// TIA Portal V16 export
// export: Created 2022-07-21T09:35:34.8398249Z, ExportSetting WithDefaults, DisplayName Totally Integrated Automation Portal, DisplayVersion V16 Update 4, DisplayName TIA Portal Version Control Interface, DisplayVersion V16 Update 2, DisplayName TIA Portal Openness, DisplayVersion V16 Update 4, DisplayName SINAMICS Startdrive Advanced, DisplayVersion V16 Update 5, DisplayName SINAMICS Startdrive G130, G150, S120, S150, SINAMICS MV, S210, DisplayVersion V16 Update 5, DisplayName SINAMICS Startdrive G110M, G120, G120C, G120D, G120P, G115D, DisplayVersion V16 Update 5, DisplayName STEP 7 Professional, DisplayVersion V16 Update 4, DisplayName STEP 7 Safety, DisplayVersion V16, DisplayName WinCC Advanced, DisplayVersion V16 Update 4
FUNCTION_BLOCK "fbGroup"   // FB700, LAD
TITLE = Group / Grupa
{ S7_Optimized_Access := 'TRUE' }
VERSION : 0.1
// stored: AutoNumber false, IsIECCheckEnabled false, IsRetainMemResEnabled false, MemoryReserve 100, SetENOAutomatically false, UDAEnableTagReadback false
   VAR_INPUT
      startDelay : Time := T#1s;   // Czas opóźnienia dla startu grupy / Start delay
      cancelEndOfSeq : Bool;   // Sygnał anulowania zatrzymania na końcu sekwencji / Cancel stop end of sequence
   END_VAR
   VAR_OUTPUT
      startup : Bool;   // Ostrzeżenie przed uruchomieniem pracy w trybie auto / Warning startup in automatic mode
   END_VAR
   VAR_IN_OUT
      group : "typeGroup";   // Grupa / Group
      extGroup : "typeGroup";   // Żądanie zewnętrzne / External request
   END_VAR
   VAR
      instTmrDlyStart { S7_SetPoint := 'True'} : TON_TIME;   // Opóźnienie dla startu grupy / Start delay
      instReset { S7_SetPoint := 'True'} : "fbReset";
      statPManual { S7_SetPoint := 'True'} : Bool;
      statPStep : Bool;
      statPAuto : Bool;
      statNSafe : Bool;
      instTmrHomeCmd { S7_SetPoint := 'True'} : TON_TIME;
   END_VAR
   VAR_TEMP   // added for the SCL form of the ladder/FBD networks
      _w1 : Bool;
      _w2 : Bool;
   END_VAR
BEGIN

REGION Network 1: Komenda "Reset"
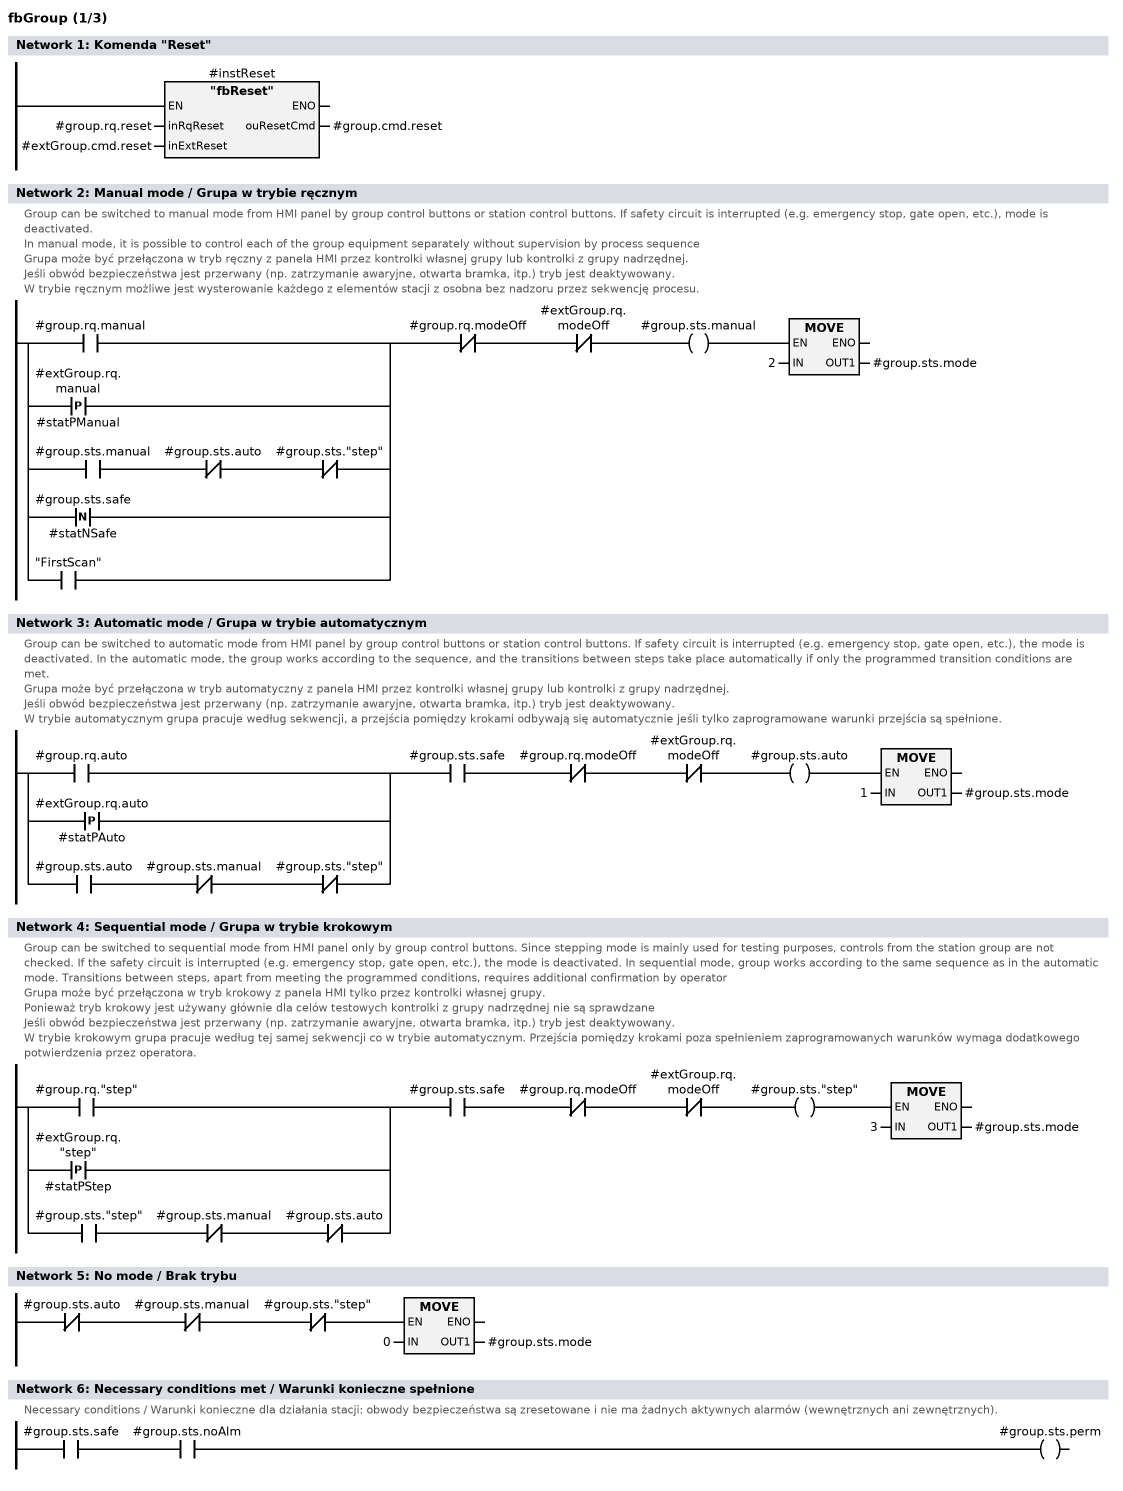
   RUNG wire#powerrail
      #instReset(inRqReset := #group.rq.reset, inExtReset := #extGroup.cmd.reset, ouResetCmd => #group.cmd.reset)
   END_RUNG
   // the same network as SCL:
   #instReset(inRqReset := #group.rq.reset, inExtReset := #extGroup.cmd.reset, ouResetCmd => #group.cmd.reset);   // "fbReset"
END_REGION

REGION Network 2: Manual mode / Grupa w trybie ręcznym
   // Group can be switched to manual mode from HMI panel by group control buttons or station control buttons. If safety circuit is interrupted (e.g. emergency stop, gate open, etc.), mode is deactivated.
   //  In manual mode, it is possible to control each of the group equipment separately without supervision by process sequence
   // Grupa może być przełączona w tryb ręczny z panela HMI przez kontrolki własnej grupy lub kontrolki z grupy nadrzędnej.
   // Jeśli obwód bezpieczeństwa jest przerwany (np. zatrzymanie awaryjne, otwarta bramka, itp.) tryb jest deaktywowany.
   // W trybie ręcznym możliwe jest wysterowanie każdego z elementów stacji z osobna bez nadzoru przez sekwencję procesu.
   RUNG wire#powerrail
      Contact( #group.rq.manual )
      wire#w1
      I_Contact( #group.rq.modeOff )
      I_Contact( #extGroup.rq.modeOff )
      Coil( #group.sts.manual )
      Move(in := 2, out1 => #group.sts.mode)
   END_RUNG
   RUNG wire#powerrail
      P_Contact(operand := #extGroup.rq.manual, bit := #statPManual)
   END_RUNG wire#w1
   RUNG wire#powerrail
      Contact( #group.sts.manual )
      I_Contact( #group.sts.auto )
      I_Contact( #group.sts."step" )
   END_RUNG wire#w1
   RUNG wire#powerrail
      N_Contact(operand := #group.sts.safe, bit := #statNSafe)
   END_RUNG wire#w1
   RUNG wire#powerrail
      Contact( "FirstScan" )
   END_RUNG wire#w1
   // the same network as SCL:
   #_w1 := #extGroup.rq.manual AND NOT #statPManual;   // rising edge of #extGroup.rq.manual
   #statPManual := #extGroup.rq.manual;
   #_w2 := NOT #group.sts.safe AND #statNSafe;   // falling edge of #group.sts.safe
   #statNSafe := #group.sts.safe;
   #group.sts.manual := (#group.rq.manual OR #_w1 OR (#group.sts.manual AND NOT #group.sts.auto AND NOT #group.sts."step") OR #_w2 OR "FirstScan") AND NOT #group.rq.modeOff AND NOT #extGroup.rq.modeOff;
   IF #group.sts.manual THEN #group.sts.mode := 2; END_IF;
END_REGION

REGION Network 3: Automatic mode / Grupa w trybie automatycznym
   // Group can be switched to automatic mode from HMI panel by group control buttons or station control buttons. If safety circuit is interrupted (e.g. emergency stop, gate open, etc.), the mode is deactivated. In the automatic mode, the group works according to the sequence, and the transitions between steps take place automatically if only the programmed transition conditions are met.
   // Grupa może być przełączona w tryb automatyczny z panela HMI przez kontrolki własnej grupy lub kontrolki z grupy nadrzędnej.
   // Jeśli obwód bezpieczeństwa jest przerwany (np. zatrzymanie awaryjne, otwarta bramka, itp.) tryb jest deaktywowany.
   // W trybie automatycznym grupa pracuje według sekwencji, a przejścia pomiędzy krokami odbywają się automatycznie jeśli tylko zaprogramowane warunki przejścia są spełnione.
   RUNG wire#powerrail
      Contact( #group.rq.auto )
      wire#w1
      Contact( #group.sts.safe )
      I_Contact( #group.rq.modeOff )
      I_Contact( #extGroup.rq.modeOff )
      Coil( #group.sts.auto )
      Move(in := 1, out1 => #group.sts.mode)
   END_RUNG
   RUNG wire#powerrail
      P_Contact(operand := #extGroup.rq.auto, bit := #statPAuto)
   END_RUNG wire#w1
   RUNG wire#powerrail
      Contact( #group.sts.auto )
      I_Contact( #group.sts.manual )
      I_Contact( #group.sts."step" )
   END_RUNG wire#w1
   // the same network as SCL:
   #_w1 := #extGroup.rq.auto AND NOT #statPAuto;   // rising edge of #extGroup.rq.auto
   #statPAuto := #extGroup.rq.auto;
   #group.sts.auto := (#group.rq.auto OR #_w1 OR (#group.sts.auto AND NOT #group.sts.manual AND NOT #group.sts."step")) AND #group.sts.safe AND NOT #group.rq.modeOff AND NOT #extGroup.rq.modeOff;
   IF #group.sts.auto THEN #group.sts.mode := 1; END_IF;
END_REGION

REGION Network 4: Sequential mode / Grupa w trybie krokowym
   // Group can be switched to sequential mode from HMI panel only by group control buttons. Since stepping mode is mainly used for testing purposes, controls from the station group are not checked. If the safety circuit is interrupted (e.g. emergency stop, gate open, etc.), the mode is deactivated. In sequential mode, group works according to the same sequence as in the automatic mode. Transitions between steps, apart from meeting the programmed conditions, requires additional confirmation by operator
   // Grupa może być przełączona w tryb krokowy z panela HMI tylko przez kontrolki własnej grupy.
   // Ponieważ tryb krokowy jest używany głównie dla celów testowych kontrolki z grupy nadrzędnej nie są sprawdzane
   // Jeśli obwód bezpieczeństwa jest przerwany (np. zatrzymanie awaryjne, otwarta bramka, itp.) tryb jest deaktywowany.
   // W trybie krokowym grupa pracuje według tej samej sekwencji co w trybie automatycznym. Przejścia pomiędzy krokami poza spełnieniem zaprogramowanych warunków wymaga dodatkowego potwierdzenia przez operatora.
   RUNG wire#powerrail
      Contact( #group.rq."step" )
      wire#w1
      Contact( #group.sts.safe )
      I_Contact( #group.rq.modeOff )
      I_Contact( #extGroup.rq.modeOff )
      Coil( #group.sts."step" )
      Move(in := 3, out1 => #group.sts.mode)
   END_RUNG
   RUNG wire#powerrail
      P_Contact(operand := #extGroup.rq."step", bit := #statPStep)
   END_RUNG wire#w1
   RUNG wire#powerrail
      Contact( #group.sts."step" )
      I_Contact( #group.sts.manual )
      I_Contact( #group.sts.auto )
   END_RUNG wire#w1
   // the same network as SCL:
   #_w1 := #extGroup.rq."step" AND NOT #statPStep;   // rising edge of #extGroup.rq."step"
   #statPStep := #extGroup.rq."step";
   #group.sts."step" := (#group.rq."step" OR #_w1 OR (#group.sts."step" AND NOT #group.sts.manual AND NOT #group.sts.auto)) AND #group.sts.safe AND NOT #group.rq.modeOff AND NOT #extGroup.rq.modeOff;
   IF #group.sts."step" THEN #group.sts.mode := 3; END_IF;
END_REGION

REGION Network 5: No mode / Brak trybu
   RUNG wire#powerrail
      I_Contact( #group.sts.auto )
      I_Contact( #group.sts.manual )
      I_Contact( #group.sts."step" )
      Move(in := 0, out1 => #group.sts.mode)
   END_RUNG
   // the same network as SCL:
   IF NOT #group.sts.auto AND NOT #group.sts.manual AND NOT #group.sts."step" THEN
       #group.sts.mode := 0;
   END_IF;
END_REGION

REGION Network 6: Necessary conditions met / Warunki konieczne spełnione
   // Necessary conditions / Warunki konieczne dla działania stacji: obwody bezpieczeństwa są zresetowane i nie ma żadnych aktywnych alarmów (wewnętrznych ani zewnętrznych).
   RUNG wire#powerrail
      Contact( #group.sts.safe )
      Contact( #group.sts.noAlm )
      Coil( #group.sts.perm )
   END_RUNG
   // the same network as SCL:
   #group.sts.perm := #group.sts.safe AND #group.sts.noAlm;
END_REGION

REGION Network 7: Ready to start / Grupa gotowa do startu
   // Group is ready to start if automatic/sequential mode is selected, necessary conditions are met, all equipment is in home position, sequence is in initial step / Grupa jest gotowa do rozpoczęcia pracy według sekwencji jeśli wybrano tryb automatyczny lub krokowy, warunki konieczne są spełnione, wszystkie elementy stacji są w pozycji bazowej i sekwencja pracy znajduje się w kroku początkowym.
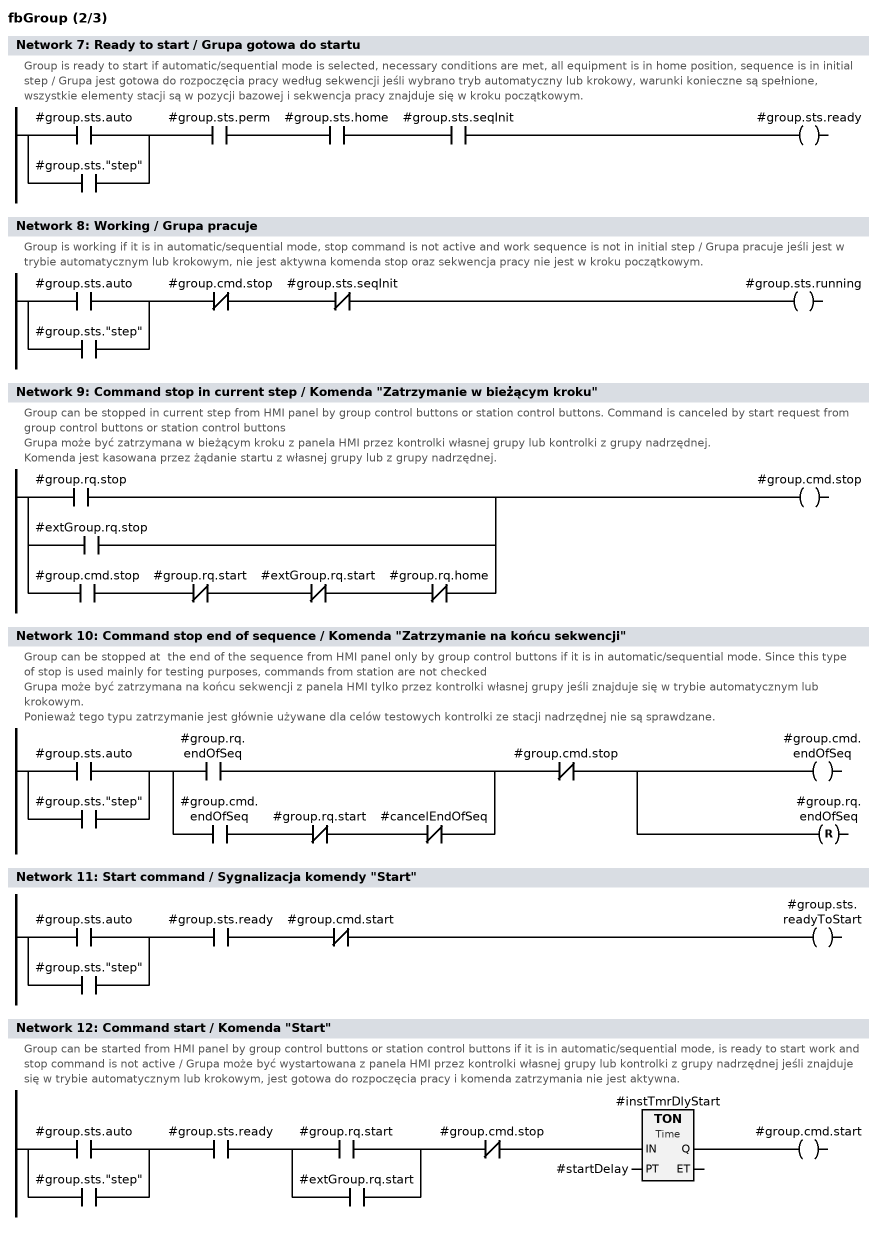
   RUNG wire#powerrail
      Contact( #group.sts.auto )
      wire#w1
      Contact( #group.sts.perm )
      Contact( #group.sts.home )
      Contact( #group.sts.seqInit )
      Coil( #group.sts.ready )
   END_RUNG
   RUNG wire#powerrail
      Contact( #group.sts."step" )
   END_RUNG wire#w1
   // the same network as SCL:
   #group.sts.ready := (#group.sts.auto OR #group.sts."step") AND #group.sts.perm AND #group.sts.home AND #group.sts.seqInit;
END_REGION

REGION Network 8: Working / Grupa pracuje
   // Group is working if it is in automatic/sequential mode, stop command is not active and work sequence is not in initial step / Grupa pracuje jeśli jest w trybie automatycznym lub krokowym, nie jest aktywna komenda stop oraz sekwencja pracy nie jest w kroku początkowym.
   RUNG wire#powerrail
      Contact( #group.sts.auto )
      wire#w1
      I_Contact( #group.cmd.stop )
      I_Contact( #group.sts.seqInit )
      Coil( #group.sts.running )
   END_RUNG
   RUNG wire#powerrail
      Contact( #group.sts."step" )
   END_RUNG wire#w1
   // the same network as SCL:
   #group.sts.running := (#group.sts.auto OR #group.sts."step") AND NOT #group.cmd.stop AND NOT #group.sts.seqInit;
END_REGION

REGION Network 9: Command stop in current step / Komenda "Zatrzymanie w bieżącym kroku"
   // Group can be stopped in current step from HMI panel by group control buttons or station control buttons. Command is canceled by start request from group control buttons or station control buttons
   // Grupa może być zatrzymana w bieżącym kroku z panela HMI przez kontrolki własnej grupy lub kontrolki z grupy nadrzędnej.
   // Komenda jest kasowana przez żądanie startu z własnej grupy lub z grupy nadrzędnej.
   RUNG wire#powerrail
      Contact( #group.rq.stop )
      wire#w1
      Coil( #group.cmd.stop )
   END_RUNG
   RUNG wire#powerrail
      Contact( #extGroup.rq.stop )
   END_RUNG wire#w1
   RUNG wire#powerrail
      Contact( #group.cmd.stop )
      I_Contact( #group.rq.start )
      I_Contact( #extGroup.rq.start )
      I_Contact( #group.rq.home )
   END_RUNG wire#w1
   // the same network as SCL:
   #group.cmd.stop := #group.rq.stop OR #extGroup.rq.stop OR (#group.cmd.stop AND NOT #group.rq.start AND NOT #extGroup.rq.start AND NOT #group.rq.home);
END_REGION

REGION Network 10: Command stop end of sequence / Komenda "Zatrzymanie na końcu sekwencji"
   // Group can be stopped at  the end of the sequence from HMI panel only by group control buttons if it is in automatic/sequential mode. Since this type of stop is used mainly for testing purposes, commands from station are not checked
   // Grupa może być zatrzymana na końcu sekwencji z panela HMI tylko przez kontrolki własnej grupy jeśli znajduje się w trybie automatycznym lub krokowym.
   // Ponieważ tego typu zatrzymanie jest głównie używane dla celów testowych kontrolki ze stacji nadrzędnej nie są sprawdzane.
   RUNG wire#powerrail
      Contact( #group.sts.auto )
      wire#w1
      Contact( #group.rq.endOfSeq )
      wire#w2
      I_Contact( #group.cmd.stop )
      wire#w3
      Coil( #group.cmd.endOfSeq )
   END_RUNG
   RUNG wire#powerrail
      Contact( #group.sts."step" )
   END_RUNG wire#w1
   RUNG wire#w1
      Contact( #group.cmd.endOfSeq )
      I_Contact( #group.rq.start )
      I_Contact( #cancelEndOfSeq )
   END_RUNG wire#w2
   RUNG wire#w3
      R_Coil( #group.rq.endOfSeq )
   END_RUNG
   // the same network as SCL:
   #group.cmd.endOfSeq := (#group.sts.auto OR #group.sts."step") AND (#group.rq.endOfSeq OR (#group.cmd.endOfSeq AND NOT #group.rq.start AND NOT #cancelEndOfSeq)) AND NOT #group.cmd.stop;
   IF #group.cmd.endOfSeq THEN #group.rq.endOfSeq := FALSE; END_IF;
END_REGION

REGION Network 11: Start command / Sygnalizacja komendy "Start"
   RUNG wire#powerrail
      Contact( #group.sts.auto )
      wire#w1
      Contact( #group.sts.ready )
      I_Contact( #group.cmd.start )
      Coil( #group.sts.readyToStart )
   END_RUNG
   RUNG wire#powerrail
      Contact( #group.sts."step" )
   END_RUNG wire#w1
   // the same network as SCL:
   #group.sts.readyToStart := (#group.sts.auto OR #group.sts."step") AND #group.sts.ready AND NOT #group.cmd.start;
END_REGION

REGION Network 12: Command start / Komenda "Start"
   // Group can be started from HMI panel by group control buttons or station control buttons if it is in automatic/sequential mode, is ready to start work and stop command is not active / Grupa może być wystartowana z panela HMI przez kontrolki własnej grupy lub kontrolki z grupy nadrzędnej jeśli znajduje się w trybie automatycznym lub krokowym, jest gotowa do rozpoczęcia pracy i komenda zatrzymania nie jest aktywna.
   RUNG wire#powerrail
      Contact( #group.sts.auto )
      wire#w1
      Contact( #group.sts.ready )
      wire#w2
      Contact( #group.rq.start )
      wire#w3
      I_Contact( #group.cmd.stop )
      { S7_Templates := "time_type := Time" } #instTmrDlyStart.TON(pt := #startDelay, et =>)
      Coil( #group.cmd.start )
   END_RUNG
   RUNG wire#powerrail
      Contact( #group.sts."step" )
   END_RUNG wire#w1
   RUNG wire#w2
      Contact( #extGroup.rq.start )
   END_RUNG wire#w3
   // the same network as SCL:
   #instTmrDlyStart(IN := (#group.sts.auto OR #group.sts."step") AND #group.sts.ready AND (#group.rq.start OR #extGroup.rq.start) AND NOT #group.cmd.stop,   // TON
                    PT := #startDelay);
   #group.cmd.start := #instTmrDlyStart.Q;
END_REGION

REGION Network 13: Command homing / Komenda "Bazowanie stacji" (wszystkie elementy stacji do pozycji bazowej)
   // Group can be "homed" only in manual mode. Homing can be initialized from HMI panel by group control buttons or station control buttons. Command is deactivated when all equipment reach home position and sequence is in initial step
   // Grupa może być "zbazowana" tylko w trybie ręcznym.
   // Bazowanie może zostać zainicjowane z panela HMI przez kontrolki z własnej grupy lub kontrolki z grupy nadrzędnej.
   // Komenda jest deaktywowana jeśli wszystkie elementy stacji osiągną pozycję bazową i sekwencja pracy znajduje się w kroku początkowym.
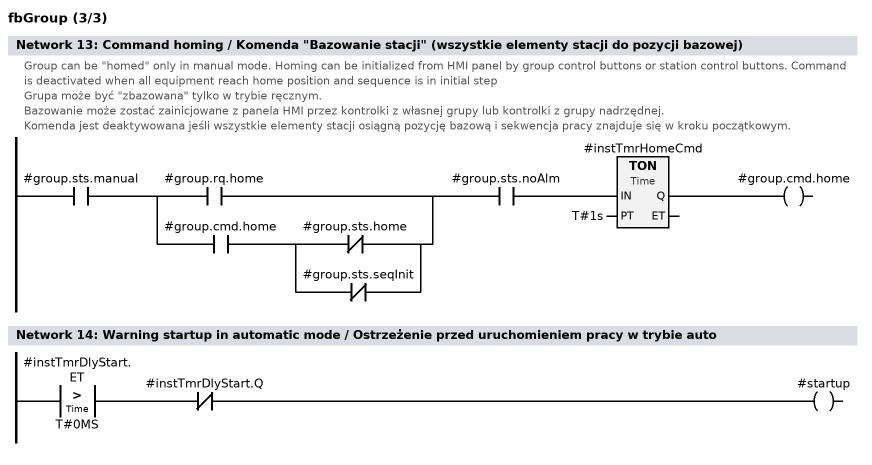
   RUNG wire#powerrail
      Contact( #group.sts.manual )
      wire#w1
      Contact( #group.rq.home )
      wire#w2
      Contact( #group.sts.noAlm )
      { S7_Templates := "time_type := Time" } #instTmrHomeCmd.TON(pt := T#1s, et =>)
      Coil( #group.cmd.home )
   END_RUNG
   RUNG wire#w1
      Contact( #group.cmd.home )
      wire#w3
      I_Contact( #group.sts.home )
   END_RUNG wire#w2
   RUNG wire#w3
      I_Contact( #group.sts.seqInit )
   END_RUNG wire#w2
   // the same network as SCL:
   #instTmrHomeCmd(IN := #group.sts.manual AND (#group.rq.home OR (#group.cmd.home AND (NOT #group.sts.home OR NOT #group.sts.seqInit))) AND #group.sts.noAlm,   // TON
                   PT := T#1s);
   #group.cmd.home := #instTmrHomeCmd.Q;
END_REGION

REGION Network 14: Warning startup in automatic mode / Ostrzeżenie przed uruchomieniem pracy w trybie auto
   RUNG wire#powerrail
      { S7_Templates := "SrcType := Time" } GT_Contact(in1 := #instTmrDlyStart.ET, in2 := T#0MS)
      I_Contact( #instTmrDlyStart.Q )
      Coil( #startup )
   END_RUNG
   // the same network as SCL:
   #startup := (#instTmrDlyStart.ET > T#0MS) AND NOT #instTmrDlyStart.Q;
END_REGION
END_FUNCTION_BLOCK
